KUKA KRL program: movement_test_lin.src, movement_test_lin.dat

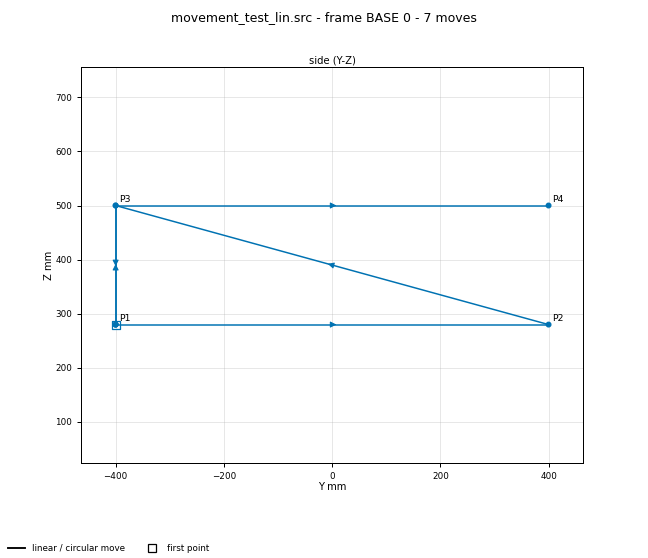
[picture p0: tool path of movement_test_lin.src in frame BASE 0, 7 of 10 moves have a stored position in this frame; points joined in program order, loops and branches not executed]
--- movement_test_lin.src ---
&ACCESS RVO
&REL 27
&PARAM DISKPATH = KRC:\R1\Program\My_Project
DEF  movement_test_lin ( )
;FOLD INI;%{PE}
  ;FOLD BASISTECH INI
    GLOBAL INTERRUPT DECL 3 WHEN $STOPMESS==TRUE DO IR_STOPM ( )
    INTERRUPT ON 3
    BAS (#INITMOV,0 )
  ;ENDFOLD (BASISTECH INI)
  ;FOLD USER INI
    ;Make your modifications here

  ;ENDFOLD (USER INI)
;ENDFOLD (INI)

;FOLD SPTP HOME Vel=100 % DEFAULT ;%{PE}
;FOLD Parameters ;%{h}
;Params IlfProvider=kukaroboter.basistech.inlineforms.movement.spline; Kuka.IsGlobalPoint=False; Kuka.PointName=HOME; Kuka.BlendingEnabled=False; Kuka.MoveDataPtpName=DEFAULT; Kuka.VelocityPtp=100; Kuka.VelocityFieldEnabled=True; Kuka.CurrentCDSetIndex=0; Kuka.MovementParameterFieldEnabled=True; IlfCommand=SPTP
;ENDFOLD
;SPTP XHOME WITH $VEL_AXIS[1] = SVEL_JOINT(100.0), $TOOL = STOOL2(FHOME), $BASE = SBASE(FHOME.BASE_NO), $IPO_MODE = SIPO_MODE(FHOME.IPO_FRAME), $LOAD = SLOAD(FHOME.TOOL_NO), $ACC_AXIS[1] = SACC_JOINT(PDEFAULT), $APO = SAPO_PTP(PDEFAULT), $GEAR_JERK[1] = SGEAR_JERK(PDEFAULT), $COLLMON_TOL_PRO[1] = USE_CM_PRO_VALUES(0)
PTP HOME                                    ;Go to Home position
;ENDFOLD

;-----------------------------------------------------------------------------
;           LINEAR MOTION - HORIZONTAL AND DIAGONAL (MIRRORED 'Z')
;-----------------------------------------------------------------------------

TraceStart("New_KSS_8.5_1.xml", "Linear_updated_sim")   ;Start recording trace with the mentioned Trace configuration

$BWDSTART = FALSE
PDAT_ACT=PPDATP
FDAT_ACT=FP
BAS (#PTP_PARAMS,100)
SET_CD_PARAMS(0)

$VEL.CP = 1                                             ;Set Cartesian velocity to 50% of the maximum value
PTP P1                                                  ;PTP movement to Point P1

$ORI_TYPE = #CONSTANT                                   ;Set Orientation of the TCP to be CONSTANT
LIN P2                                                  ;Linear movement to Point P2
$ORI_TYPE = #JOINT                                      ;Set Orientation of the TCP to be JOINT type
LIN P3                                                  ;Linear movement to Point P3
LIN P4                                                  ;Linear movement to Point P4

TraceStop()

PTP HOME                                                ;Go to Home position

;-----------------------------------------------------------------------------
;                    LINEAR VERTICAL MOTION
;-----------------------------------------------------------------------------
TraceStart("New_KSS_8.5_1.xml", "Linear_vertical_sim")  ;Start recording trace with the mentioned Trace configuration

$VEL.CP = 1                                             ;Set Cartesian velocity to 50% of the maximum value
PTP P1                                                  ;PTP movement to Point P1

$ORI_TYPE = #JOINT                                      ;Set Orientation of the TCP to be JOINT type
LIN P3                                                  ;Linear movement to Point P3

WAIT SEC 2                                              ;Set a delay of 2 seconds

LIN P1                                                  ;Linear movement to Point P1

PTP HOME                                                ;Go to Home position

TraceStop()

END

--- movement_test_lin.dat ---
&ACCESS RVO
&REL 27
&PARAM DISKPATH = KRC:\R1\Program\My_Project
DEFDAT  MOVEMENT_TEST_LIN
;FOLD EXTERNAL DECLARATIONS;%{PE}%MKUKATPBASIS,%CEXT,%VCOMMON,%P
;FOLD BASISTECH EXT;%{PE}%MKUKATPBASIS,%CEXT,%VEXT,%P
EXT  BAS (BAS_COMMAND  :IN,REAL  :IN )
DECL INT SUCCESS
;ENDFOLD (BASISTECH EXT)
;FOLD USER EXT;%{E}%MKUKATPUSER,%CEXT,%VEXT,%P
;Make your modifications here

DECL E6AXIS HOME={A1 0.0,A2 -110.000,A3 110.000,A4 0.0,A5 0.0,A6 0.0}          ;Home Position

DECL PDAT PPDATP={VEL 10.000,ACC 100.000,APO_DIST 100.000,APO_MODE #CDIS,GEAR_JERK 100.000,EXAX_IGN 0}     ;Set the kinematic values such as max velocity, max acceleration, etc
DECL FDAT FP={TOOL_NO 14,BASE_NO 0,IPO_FRAME #BASE,POINT2[] " ",TQ_STATE FALSE}                            ;Set the tool and base for coordinate transformation

DECL E6POS P1={X 350.000,Y -400.000,Z 280.000,A -0.9,B 30.76,C -3.04,S 6,T 50}      ;Point P1
DECL E6POS P2={X 350.000,Y 400.000,Z 280.000,A -0.9,B 30.76,C -3.04,S 6,T 27}       ;Point P2
DECL E6POS P3={X 350.000,Y -400.000,Z 500.000,A -0.9,B 30.76,C -3.04,S 6,T 50}      ;Point P3
DECL E6POS P4={X 350.000,Y 400.000,Z 500.000,A -0.9,B 30.76,C -3.04,S 6,T 27}       ;Point P4

;ENDFOLD (USER EXT)
;ENDFOLD (EXTERNAL DECLARATIONS)
ENDDAT
